FUNCTION_BLOCK FB_Sequencer_Test EXTENDS FB_TestSuite
VAR_INPUT
END_VAR
VAR_OUTPUT
END_VAR
VAR
END_VAR

OnAbort();
RunGetsCalled();
CurrentStep();

METHOD CurrentStep
VAR
	sequencer : Sequencer(0);
	Command : PLCOpenCommand();
	output_step : UDINT;
END_VAR
TEST('CurrentStep');
	output_step := sequencer.CurrentStep;
	AssertEquals_UDINT(Expected := 0, Actual := output_step, 'Current step shall default to 0');
	sequencer.requestStep(2);
	sequencer.Run();
	output_step := sequencer.CurrentStep;
	AssertEquals_UDINT(Expected := 2, Actual := output_step, 'Current step expected to be 2');
TEST_FINISHED();
END_METHOD

METHOD OnAbort
VAR
	sequencer : Sequencer(0);
	outputVal : BOOL;
END_VAR
TEST('SequenceOnError');
	sequencer.sequenceError(0, 'Test Error');
	sequencer.Run();
	outputVal := sequencer.onError(1);
	
	AssertTrue(Condition := outputVal, Message := 'This is not a real test');
TEST_FINISHED();
END_METHOD

METHOD OnEntry
VAR_INPUT
END_VAR
TEST('OnEntry');

TEST_FINISHED();
END_METHOD

METHOD OnSuccess
VAR_INPUT
	sequencer : Sequencer(0);
END_VAR
TEST('OnSuccess');

	//sequencer.i_sequence.activeTasks
	// next step negative
	//sequencer.setNextStep(-1);
	//sequencer.onSuccess(-1);
	
	// next step >= 0


TEST_FINISHED();
END_METHOD

METHOD RequestStep
VAR_INPUT
END_VAR
TEST('NextStep');
//	sequencer.sequenceError(0, 'Test Error');
//	sequencer.Run();
//	sequencer.requestStep(1);
//	sequencer.CurrentStep := 0;
//	sequencer.Run();
	
//	outputVal := sequencer.onError(1);
	
//	AssertTrue(Condition := outputVal, Message := 'This is not a real test');
TEST_FINISHED();
END_METHOD

METHOD RunGetsCalled
VAR
	sequencer : Sequencer(0);
END_VAR
TEST('RunGetsCalled');
	sequencer.Run();
	AssertTrue(Condition := FALSE, Message := 'False Failure');
TEST_FINISHED();
END_METHOD

METHOD Start
VAR
	sequencer : Sequencer(0);
	output : BOOL;
END_VAR
TEST('Start');
	// activeTasks.Start) = 0
	// TODO
	
	//output := sequencer.i_sequence.startStep
	
	

TEST_FINISHED();
END_METHOD

END_FUNCTION_BLOCK

(* stored: Version 1.1.0.1, ProductVersion 3.1.4024.12
   POU FB_Sequencer_Test: Id {5528d32b-0dad-48bc-b63b-5f76dadd2ea9}, SpecialFunc None
   Method CurrentStep: Id {00c73c39-e570-45cb-8831-bed7304ddd26}
   Method OnAbort: Id {756190d0-8aa4-4061-8aca-7e61a0ad15cd}
   Method OnEntry: Id {3a0279ba-27ed-47d6-a39c-8c9f7c30b3c2}
   Method OnSuccess: Id {6a55c547-d864-42a2-86db-036e6aa1ad13}
   Method RequestStep: Id {b1880163-8808-4d23-8c10-95b3003a52e2}
   Method RunGetsCalled: Id {66dae229-dddb-4b20-8682-f3a53ce457fd}
   Method Start: Id {3d524a28-168c-402c-a8b1-706368e2797f} *)
